TYPE st_WarehouseLayer :
STRUCT
	bForward		:	BOOL;
	bBackward		:	BOOL;
	stStatus		:	st_LayerStatus;
END_STRUCT
END_TYPE

(* stored: Version 1.1.0.1, ProductVersion 3.1.4024.13
   DUT st_WarehouseLayer: Id {9ddda4a4-8968-44e3-a9e4-47b44cd53990} *)
